RoboDK station: Scooby_and_CRX10.rdk

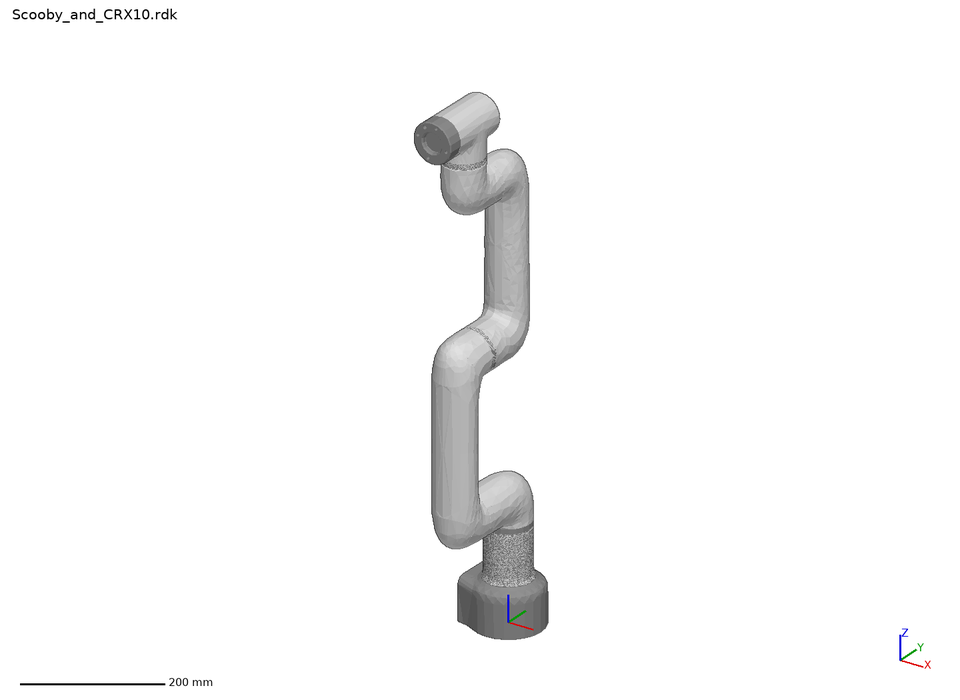
[picture v0: the station drawn from its stored meshes, robots at their saved joint values, targets as dots, program paths as lines]
Station Scooby_and_CRX10 (saved by RoboDK 5.5.4). Poses are relative to the parent item; angles as X-Y-Z fixed-axis rotations.
Station parameters (name, value as stored): LIN64
  - frame Elephant Robotics myCobot Pro-600 Base at (0, 0, 0) mm
    - robot Elephant Robotics myCobot Pro-600: 6 axes
        modified DH rows (alpha deg, a mm, theta deg, d mm): 0, 0, 0, 199.34; 90, 0, 0, 0; 0, 250, 0, 0; 0, 250, 180, 108; -90, 0, 0, 109.1; 90, 0, 0, 75.86
        joint limits [-180, -270, -150, -260, -168, -174] to [180, 90, 150, 80, 168, 174]; home [0, -90, 0, -90, 0, 0]; saved at [0, -90, 0, -90, 0, 0]
  - frame Frame 2 at (600, 0, 0) mm
